PROGRAM P5_06_Trends
VAR
END_VAR

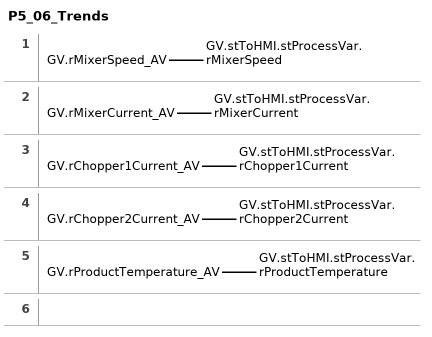
// NETWORK 1
GV.stToHMI.stProcessVar.rMixerSpeed := GV.rMixerSpeed_AV;

// NETWORK 2
GV.stToHMI.stProcessVar.rMixerCurrent := GV.rMixerCurrent_AV;

// NETWORK 3
GV.stToHMI.stProcessVar.rChopper1Current := GV.rChopper1Current_AV;

// NETWORK 4
GV.stToHMI.stProcessVar.rChopper2Current := GV.rChopper2Current_AV;

// NETWORK 5
GV.stToHMI.stProcessVar.rProductTemperature := GV.rProductTemperature_AV;

// NETWORK 6

END_PROGRAM

(* stored: Version 1.1.0.1
   POU P5_06_Trends: Id {d492406f-4b02-4ad9-938d-8e94b9df5751}, SpecialFunc None *)
